// TwinCAT 3 PLC project Untitled1
// ProgramVersion: 3.1.4023.0
// libraries:
//   Tc2_Standard, * (Beckhoff Automation GmbH)
//   Tc2_System, * (Beckhoff Automation GmbH)
//   Tc3_Module, * (Beckhoff Automation GmbH)
//   VisuSymbols,3.5.10.0,System
// project tree:
//   / PlcTask.TcTTO, 视图管理器.TcVMO (not stored)
//   POUs/ FB_A10.TcPOU, FB_Generic.TcPOU, MAIN.TcPOU
//   VISUs/ visu_main.TcVIS
// real-time tasks:
//   TASK PlcTask: cycle T#10ms, priority 20, ADS port 350

CONFIGURATION Untitled1
    RESOURCE PLC ON TwinCAT3
        TASK PlcTask(INTERVAL := T#10ms, PRIORITY := 20);
        PROGRAM MAIN WITH PlcTask : MAIN;
    END_RESOURCE
END_CONFIGURATION

// ---- POUs/MAIN.TcPOU
PROGRAM MAIN
VAR
END_VAR

END_PROGRAM

// ---- POUs/FB_A10.TcPOU
FUNCTION_BLOCK FB_A10
VAR_INPUT
END_VAR
VAR_OUTPUT
END_VAR
VAR
END_VAR

METHOD M_Abort : BOOL
VAR_INPUT
END_VAR
END_METHOD

METHOD M_Execute : BOOL
VAR_INPUT
END_VAR
END_METHOD

METHOD M_reset : BOOL
VAR_INPUT
END_VAR
//////////////////////reset all error here////////////////////////////
END_METHOD

END_FUNCTION_BLOCK

// ---- POUs/FB_Generic.TcPOU
FUNCTION_BLOCK FB_Generic
VAR_INPUT
END_VAR
VAR_OUTPUT
END_VAR
VAR
END_VAR

METHOD M_reset : BOOL
VAR_INPUT
END_VAR
END_METHOD

END_FUNCTION_BLOCK

// ---- VISUs/visu_main.TcVIS
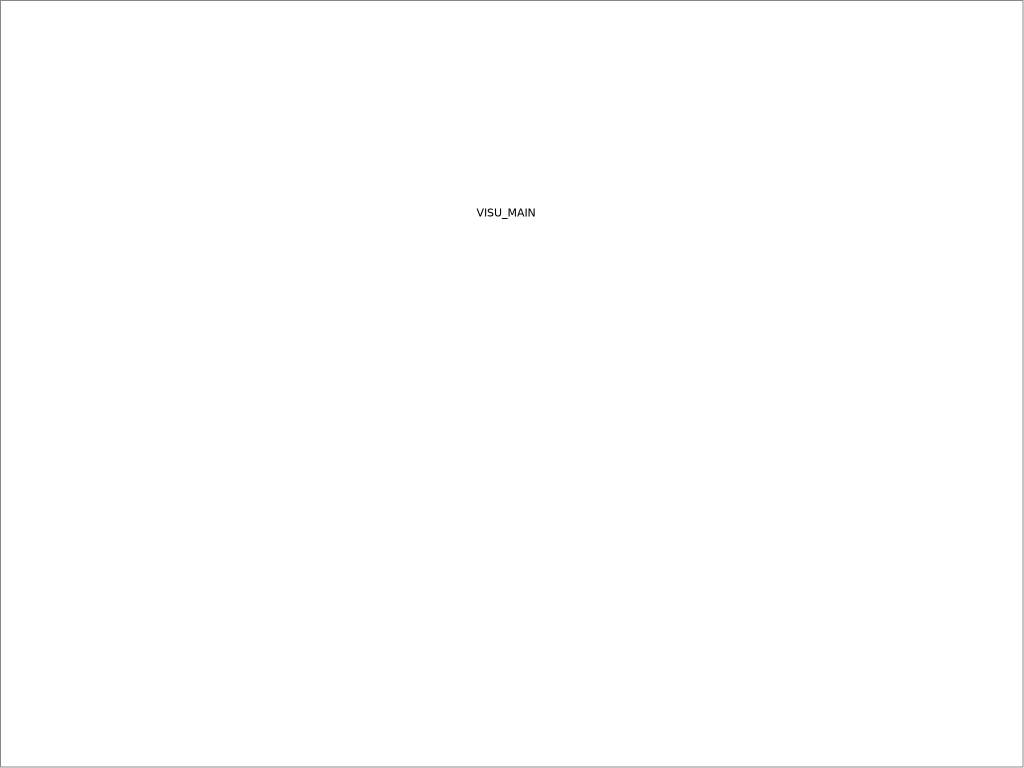
VISUALIZATION visu_main  // 1024x768
    Label (431,198 150x30), "VISU_MAIN"
END_VISUALIZATION
